// Mitsubishi GX Works2 project: LRI - PLC - AULA 7   PLC: Q00J

PROGRAM MAIN
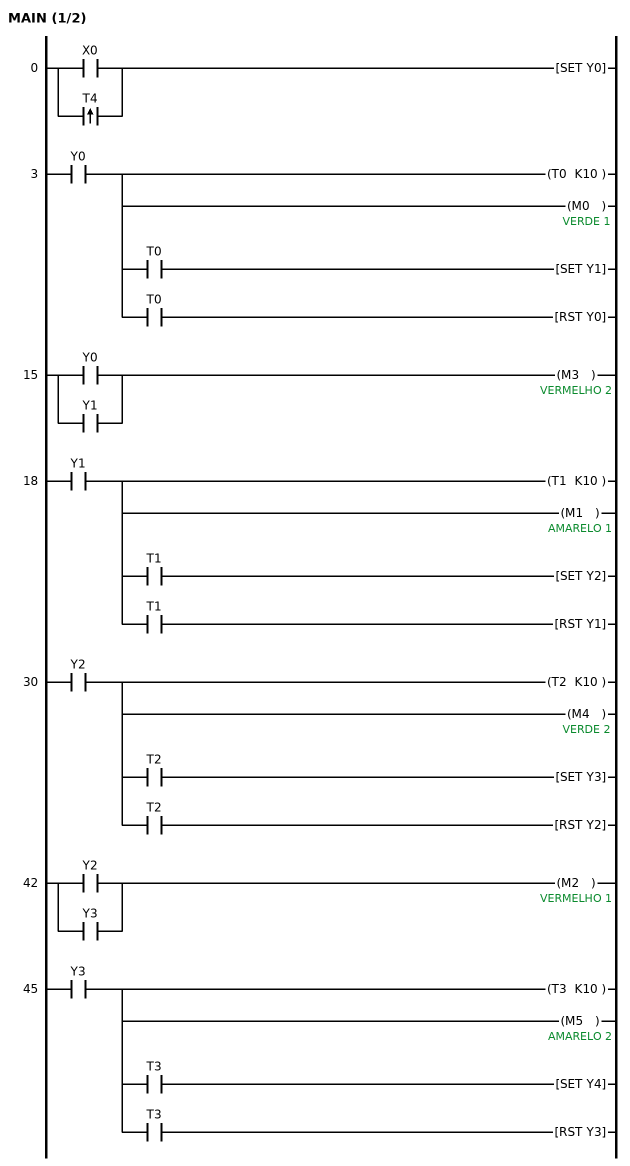
0     LD      X0
      ORP     T4
      SET     Y0
3     LD      Y0
      OUT     T0 K10
      OUT     M0  ; VERDE 1
      MPS
      AND     T0
      SET     Y1
      MPP
      AND     T0
      RST     Y0
15    LD      Y0
      OR      Y1
      OUT     M3  ; VERMELHO 2
18    LD      Y1
      OUT     T1 K10
      OUT     M1  ; AMARELO 1
      MPS
      AND     T1
      SET     Y2
      MPP
      AND     T1
      RST     Y1
30    LD      Y2
      OUT     T2 K10
      OUT     M4  ; VERDE 2
      MPS
      AND     T2
      SET     Y3
      MPP
      AND     T2
      RST     Y2
42    LD      Y2
      OR      Y3
      OUT     M2  ; VERMELHO 1
45    LD      Y3
      OUT     T3 K10
      OUT     M5  ; AMARELO 2
      MPS
      AND     T3
      SET     Y4
      MPP
      AND     T3
      RST     Y3
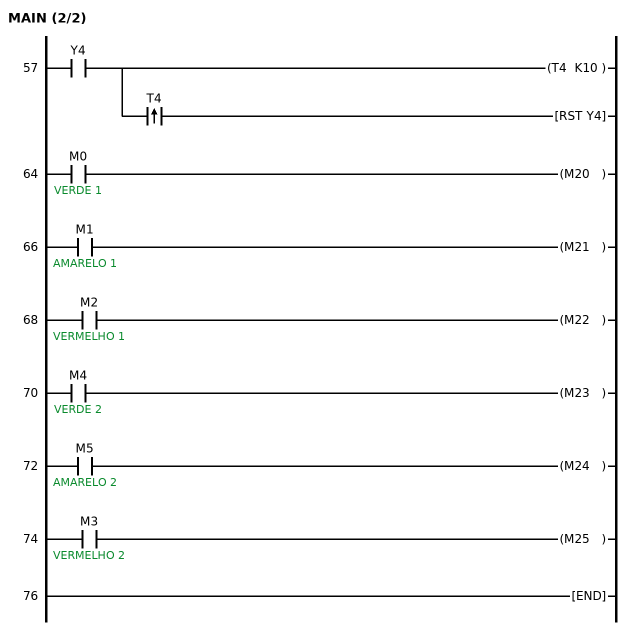
57    LD      Y4
      OUT     T4 K10
      ANDP    T4
      RST     Y4
64    LD      M0  ; VERDE 1
      OUT     M20
66    LD      M1  ; AMARELO 1
      OUT     M21
68    LD      M2  ; VERMELHO 1
      OUT     M22
70    LD      M4  ; VERDE 2
      OUT     M23
72    LD      M5  ; AMARELO 2
      OUT     M24
74    LD      M3  ; VERMELHO 2
      OUT     M25
76    END
END_PROGRAM
